Staubli VAL3: fold.pgx

program fold(string x_sDirection, num x_nEdge)
  local num l_nDim[2]
begin

  if x_sDirection == "x"
    // 0123456 7 891011121314
    call util:extractGrid(nGrid,1,0,x_nEdge-1, nLeftMatrix)
    call util:extractGrid(nGrid,1,size(nGrid,1)-1,x_nEdge+1, nRightMatrix)
  else
    call util:extractGrid(nGrid,2,0,x_nEdge-1, nLeftMatrix)
    call util:extractGrid(nGrid,2,size(nGrid,2)-1,x_nEdge+1, nRightMatrix)
  endIf

  call mat:add(nLeftMatrix, nRightMatrix, nGrid)

  // Set to one, if addition will give results > 1
  for l_nDim[0] = 0 to size(nGrid,1)-1
    for l_nDim[1] = 0 to size(nGrid,2) -1
      if nGrid[l_nDim[0], l_nDim[1]] > 1
        nGrid[l_nDim[0], l_nDim[1]] = 1
      endIf
    endFor
  endFor


end
